// TIA Portal V20 export
DATA_BLOCK "FC_Traffic_Lights_DB"   // DB3
// stored: InstanceOfName FC_Traffic_Lights, InstanceOfType FB
"FC_Traffic_Lights"
   // VAR
   //    "Timer" { S7_SetPoint := 'True'} : TON_TIME;
   // END_VAR
BEGIN
END_DATA_BLOCK
